  966 = 'S6_Warnings Default 966' | German: 'S6_Warnings German 966' | French: 'S6_Warnings French 966'
  967 = 'S6_Warnings Default 967' | German: 'S6_Warnings German 967' | French: 'S6_Warnings French 967'
  968 = 'S6_Warnings Default 968' | German: 'S6_Warnings German 968' | French: 'S6_Warnings French 968'
  969 = 'S6_Warnings Default 969' | German: 'S6_Warnings German 969' | French: 'S6_Warnings French 969'
  970 = 'S6_Warnings Default 970' | German: 'S6_Warnings German 970' | French: 'S6_Warnings French 970'
  971 = 'S6_Warnings Default 971' | German: 'S6_Warnings German 971' | French: 'S6_Warnings French 971'
  972 = 'S6_Warnings Default 972' | German: 'S6_Warnings German 972' | French: 'S6_Warnings French 972'
  973 = 'S6_Warnings Default 973' | German: 'S6_Warnings German 973' | French: 'S6_Warnings French 973'
  974 = 'S6_Warnings Default 974' | German: 'S6_Warnings German 974' | French: 'S6_Warnings French 974'
  975 = 'S6_Warnings Default 975' | German: 'S6_Warnings German 975' | French: 'S6_Warnings French 975'
  976 = 'S6_Warnings Default 976' | German: 'S6_Warnings German 976' | French: 'S6_Warnings French 976'
  977 = 'S6_Warnings Default 977' | German: 'S6_Warnings German 977' | French: 'S6_Warnings French 977'
  978 = 'S6_Warnings Default 978' | German: 'S6_Warnings German 978' | French: 'S6_Warnings French 978'
  979 = 'S6_Warnings Default 979' | German: 'S6_Warnings German 979' | French: 'S6_Warnings French 979'
  980 = 'S6_Warnings Default 980' | German: 'S6_Warnings German 980' | French: 'S6_Warnings French 980'
  981 = 'S6_Warnings Default 981' | German: 'S6_Warnings German 981' | French: 'S6_Warnings French 981'
  982 = 'S6_Warnings Default 982' | German: 'S6_Warnings German 982' | French: 'S6_Warnings French 982'
  983 = 'S6_Warnings Default 983' | German: 'S6_Warnings German 983' | French: 'S6_Warnings French 983'
  984 = 'S6_Warnings Default 984' | German: 'S6_Warnings German 984' | French: 'S6_Warnings French 984'
  985 = 'S6_Warnings Default 985' | German: 'S6_Warnings German 985' | French: 'S6_Warnings French 985'
  986 = 'S6_Warnings Default 986' | German: 'S6_Warnings German 986' | French: 'S6_Warnings French 986'
  987 = 'S6_Warnings Default 987' | German: 'S6_Warnings German 987' | French: 'S6_Warnings French 987'
  988 = 'S6_Warnings Default 988' | German: 'S6_Warnings German 988' | French: 'S6_Warnings French 988'
  989 = 'S6_Warnings Default 989' | German: 'S6_Warnings German 989' | French: 'S6_Warnings French 989'
  990 = 'S6_Warnings Default 990' | German: 'S6_Warnings German 990' | French: 'S6_Warnings French 990'
  991 = 'S6_Warnings Default 991' | German: 'S6_Warnings German 991' | French: 'S6_Warnings French 991'
  992 = 'S6_Warnings Default 992' | German: 'S6_Warnings German 992' | French: 'S6_Warnings French 992'
  993 = 'S6_Warnings Default 993' | German: 'S6_Warnings German 993' | French: 'S6_Warnings French 993'
  994 = 'S6_Warnings Default 994' | German: 'S6_Warnings German 994' | French: 'S6_Warnings French 994'
  995 = 'S6_Warnings Default 995' | German: 'S6_Warnings German 995' | French: 'S6_Warnings French 995'
  996 = 'S6_Warnings Default 996' | German: 'S6_Warnings German 996' | French: 'S6_Warnings French 996'
  997 = 'S6_Warnings Default 997' | German: 'S6_Warnings German 997' | French: 'S6_Warnings French 997'
  998 = 'S6_Warnings Default 998' | German: 'S6_Warnings German 998' | French: 'S6_Warnings French 998'
  999 = 'S6_Warnings Default 999' | German: 'S6_Warnings German 999' | French: 'S6_Warnings French 999'
  1000 = 'S6_Warnings Default 1000' | German: 'S6_Warnings German 1000' | French: 'S6_Warnings French 1000'
   = ''
END_TEXTLIST

(* stored: Version 1.1.0.1, ProductVersion 3.1.4024.12
   TextList S6_Warnings: Id {bfea007b-bd7b-4ff5-b45b-ddb2a0822c9a} *)
